FUNCTION_BLOCK FB_Gripper
VAR_INPUT
	bAirSupply	: BOOL;
	stCtrl		: Tc3_TcForms.ST_SetResetCtrl;
END_VAR
VAR_OUTPUT
	stState		: Tc3_TcForms.ST_SetResetState;
END_VAR
VAR
	rsGripper			: RS;
	tonGripper			: TON;
	tofGripper			: TOF;
	tonError			: TON;
	rtErrorAck			: R_TRIG;
END_VAR

rsGripper(SET:=stCtrl.bSet,RESET1:=stCtrl.bReset,Q1=>stState.bBusy);
tonGripper(IN:=rsGripper.Q1 AND bAirSupply,PT:=T#1S);
tofGripper(IN:=rsGripper.Q1 AND bAirSupply,PT:=T#1S);
stState.bOn := tonGripper.Q;
stState.bOff := NOT tofGripper.Q;
tonError(IN:=(stState.bBusy AND stState.bOff) OR (NOT stState.bBusy AND stState.bOn),PT:=T#2S,Q=>stState.bError);
stState.bDone := stCtrl.bSet OR stCtrl.bReset;
rtErrorAck(CLK:=stState.bDone);
IF rtErrorAck.Q THEN
	tonError(IN:=FALSE);
END_IF

END_FUNCTION_BLOCK

(* stored: Version 1.1.0.1, ProductVersion 3.1.4024.15
   POU FB_Gripper: Id {37db5731-0918-4f96-baf8-829fb750b563}, SpecialFunc None *)
